// TIA Portal V19 export
DATA_BLOCK "LB131"   // DB114
// stored: InstanceOfName ButtonsSafe_LB131, InstanceOfType FB
"ButtonsSafe_LB131"
   // VAR_INPUT
   //    Reset_OthersPBs_Activation_IN : Bool;
   // END_VAR
   // VAR_OUTPUT
   //    Reset_OthersPBs_Activation_OUT : Bool;
   // END_VAR
   // VAR
   //    i : Int;
   //    iOperation : Int;
   //    iConcurrentOperation : Int;
   //    SettingWriteDone { S7_SetPoint := 'True'} : Bool;
   //    PbPanel { S7_SetPoint := 'True'} : "Buttons2Hands";
   //    PB : Struct
   //       ResetAlarms : Bool;
   //       Decoiler_Fwd : Bool;
   //       Decoiler_Bwd : Bool;
   //       SnubberLift_Up : Bool;
   //       SnubberLift_Down : Bool;
   //       SnubberRoll_Fwd : Bool;
   //       SnubberRoll_Bwd : Bool;
   //       PeelerLift_Up : Bool;
   //       PeelerLift_Down : Bool;
   //       PeelerExtension_Fwd : Bool;
   //       PeelerExtension_Bwd : Bool;
   //       Straightner_Fwd : Bool;
   //       Straightner_Bwd : Bool;
   //    END_STRUCT;
   // END_VAR
BEGIN
END_DATA_BLOCK
